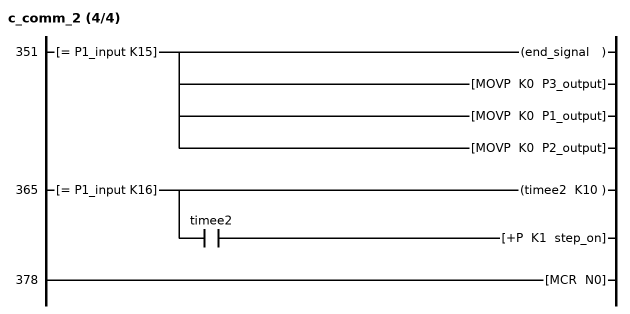
[picture p24: ladder of c_comm_2, rungs at steps 351 to 378]
351   LD=     P1_input K15
      OUT     end_signal
      MOVP    K0 P3_output
      MOVP    K0 P1_output
      MOVP    K0 P2_output
365   LD=     P1_input K16
      OUT     timee2 K10
      AND     timee2
      +P      K1 step_on
378   MCR     N0
END_FUNCTION_BLOCK

FUNCTION_BLOCK c_comm_3
VAR_INPUT
  P1_input : INT;
  P2_input : INT;
  P3_input : INT;
END_VAR
VAR_IN_OUT
  step_on : INT;
END_VAR
VAR_INPUT
  position : INT;
END_VAR
VAR
  p2_buff : INT;
END_VAR
VAR_OUTPUT
  P1_output : INT;
  P2_output : INT;
  P3_output : INT;
END_VAR
VAR_IN_OUT
  end_step_01 : INT;
END_VAR
VAR_OUTPUT
  end_signal : BOOL;
END_VAR
VAR
  mc_1234 : BOOL;
  line1_10_buff : INT;
  line2_10_buff : INT;
END_VAR
VAR_OUTPUT
  next_signal : BOOL;
END_VAR
VAR
  next_signal_01 : BOOL;
  next_signal_03 : BOOL;
  next_signal_04 : BOOL;
  next_signal_05 : BOOL;
  next_signal_06 : BOOL;
  next_signal_07 : BOOL;
  next_signal_08 : BOOL;
  punch1 : BOOL;
  punch3 : BOOL;
  punch4 : BOOL;
  punch5 : BOOL;
  punch6 : BOOL;
  punch7 : BOOL;
END_VAR
VAR_OUTPUT
  punch : BOOL;
END_VAR
VAR
  punch2 : BOOL;
  timee : TIMER;
  timee2 : TIMER;
END_VAR
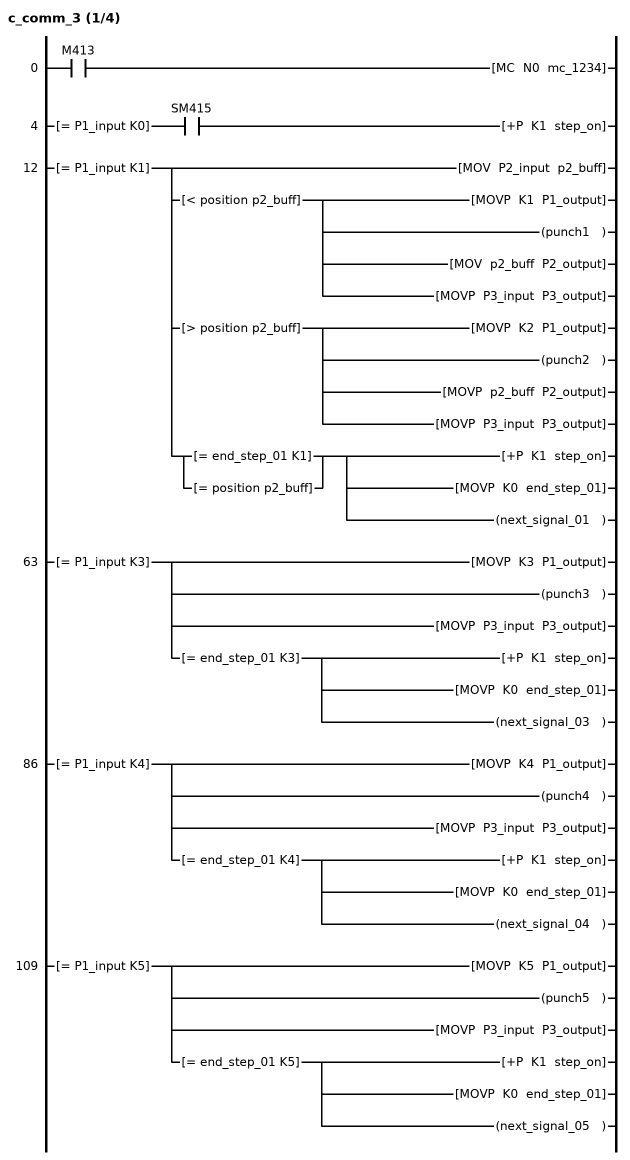
0     LD      M413
      MC      N0 mc_1234
4     LD=     P1_input K0
      AND     SM415
      +P      K1 step_on
12    LD=     P1_input K1
      MOV     P2_input p2_buff
      MPS
      AND<    position p2_buff
      MOVP    K1 P1_output
      OUT     punch1
      MOV     p2_buff P2_output
      MOVP    P3_input P3_output
      MRD
      AND>    position p2_buff
      MOVP    K2 P1_output
      OUT     punch2
      MOVP    p2_buff P2_output
      MOVP    P3_input P3_output
      MPP
      LD=     end_step_01 K1
      OR=     position p2_buff
      ANB
      +P      K1 step_on
      MOVP    K0 end_step_01
      OUT     next_signal_01
63    LD=     P1_input K3
      MOVP    K3 P1_output
      OUT     punch3
      MOVP    P3_input P3_output
      AND=    end_step_01 K3
      +P      K1 step_on
      MOVP    K0 end_step_01
      OUT     next_signal_03
86    LD=     P1_input K4
      MOVP    K4 P1_output
      OUT     punch4
      MOVP    P3_input P3_output
      AND=    end_step_01 K4
      +P      K1 step_on
      MOVP    K0 end_step_01
      OUT     next_signal_04
109   LD=     P1_input K5
      MOVP    K5 P1_output
      OUT     punch5
      MOVP    P3_input P3_output
      AND=    end_step_01 K5
      +P      K1 step_on
      MOVP    K0 end_step_01
      OUT     next_signal_05
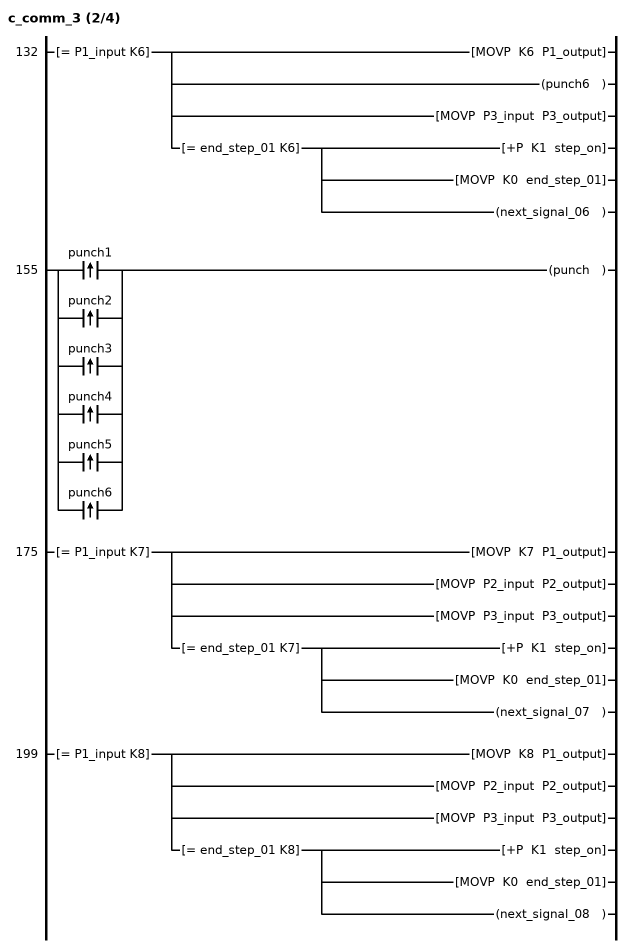
132   LD=     P1_input K6
      MOVP    K6 P1_output
      OUT     punch6
      MOVP    P3_input P3_output
      AND=    end_step_01 K6
      +P      K1 step_on
      MOVP    K0 end_step_01
      OUT     next_signal_06
155   LDP     punch1
      ORP     punch2
      ORP     punch3
      ORP     punch4
      ORP     punch5
      ORP     punch6
      OUT     punch
175   LD=     P1_input K7
      MOVP    K7 P1_output
      MOVP    P2_input P2_output
      MOVP    P3_input P3_output
      AND=    end_step_01 K7
      +P      K1 step_on
      MOVP    K0 end_step_01
      OUT     next_signal_07
199   LD=     P1_input K8
      MOVP    K8 P1_output
      MOVP    P2_input P2_output
      MOVP    P3_input P3_output
      AND=    end_step_01 K8
      +P      K1 step_on
      MOVP    K0 end_step_01
      OUT     next_signal_08
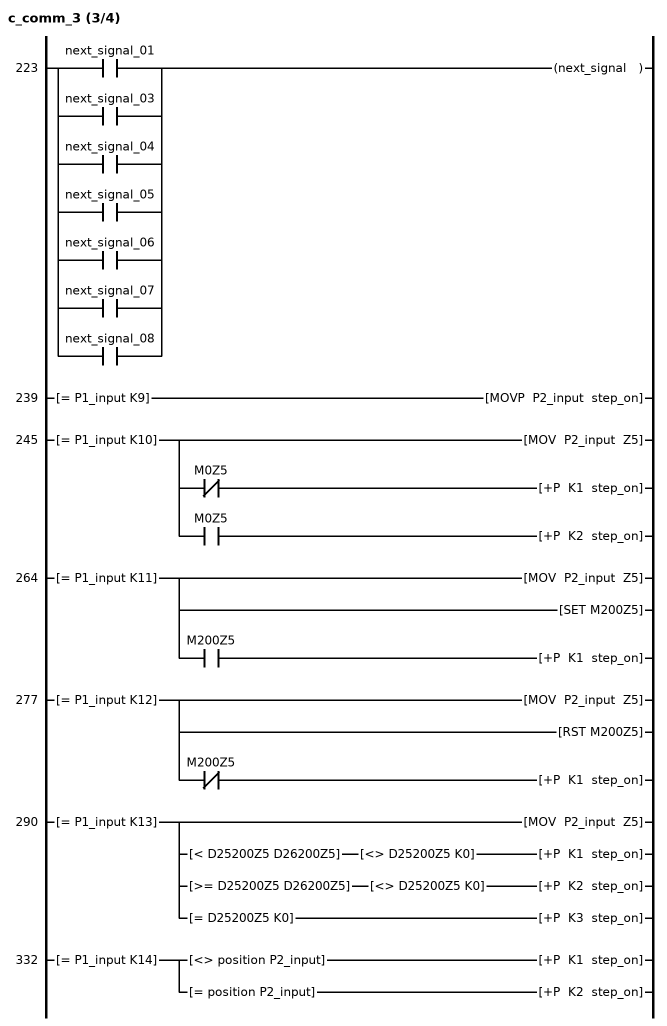
223   LD      next_signal_01
      OR      next_signal_03
      OR      next_signal_04
      OR      next_signal_05
      OR      next_signal_06
      OR      next_signal_07
      OR      next_signal_08
      OUT     next_signal
239   LD=     P1_input K9
      MOVP    P2_input step_on
245   LD=     P1_input K10
      MOV     P2_input Z5
      MPS
      ANI     M0Z5
      +P      K1 step_on
      MPP
      AND     M0Z5
      +P      K2 step_on
264   LD=     P1_input K11
      MOV     P2_input Z5
      SET     M200Z5
      AND     M200Z5
      +P      K1 step_on
277   LD=     P1_input K12
      MOV     P2_input Z5
      RST     M200Z5
      ANI     M200Z5
      +P      K1 step_on
290   LD=     P1_input K13
      MOV     P2_input Z5
      MPS
      AND<    D25200Z5 D26200Z5
      AND<>   D25200Z5 K0
      +P      K1 step_on
      MRD
      AND>=   D25200Z5 D26200Z5
      AND<>   D25200Z5 K0
      +P      K2 step_on
      MPP
      AND=    D25200Z5 K0
      +P      K3 step_on
332   LD=     P1_input K14
      MPS
      AND<>   position P2_input
      +P      K1 step_on
      MPP
      AND=    position P2_input
      +P      K2 step_on
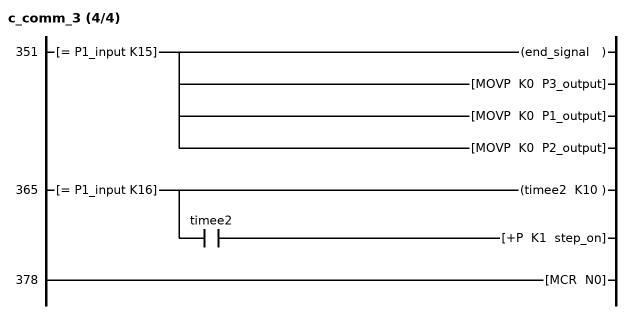
351   LD=     P1_input K15
      OUT     end_signal
      MOVP    K0 P3_output
      MOVP    K0 P1_output
      MOVP    K0 P2_output
365   LD=     P1_input K16
      OUT     timee2 K10
      AND     timee2
      +P      K1 step_on
378   MCR     N0
END_FUNCTION_BLOCK

PROGRAM carrier_01
VAR
  c_comm_1 : c_comm_1;
END_VAR
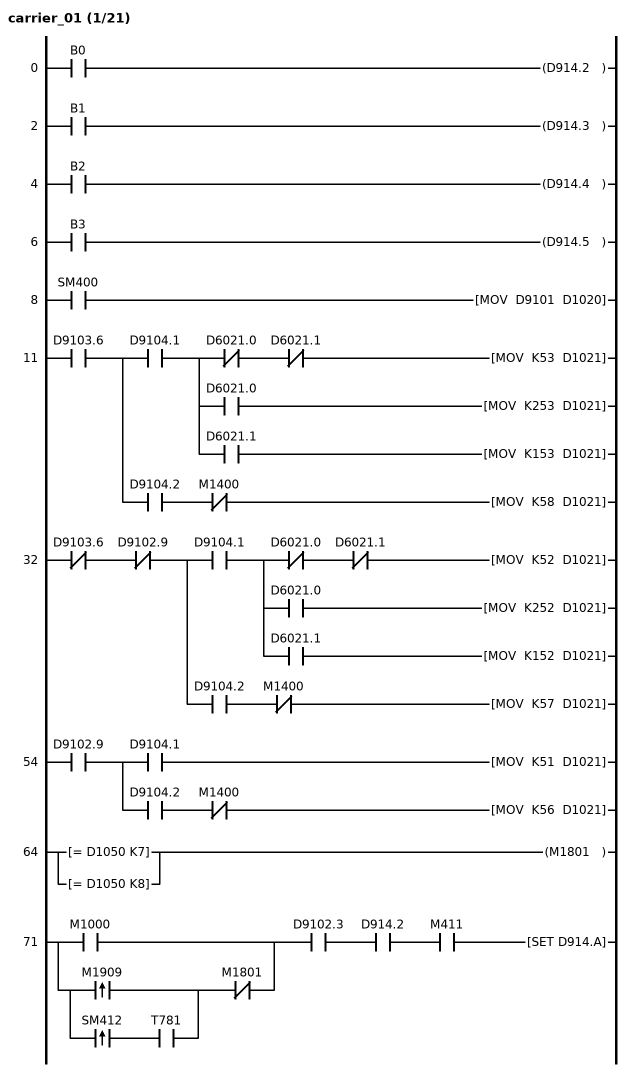
0     LD      B0
      OUT     D914.2
2     LD      B1
      OUT     D914.3
4     LD      B2
      OUT     D914.4
6     LD      B3
      OUT     D914.5
8     LD      SM400
      MOV     D9101 D1020
11    LD      D9103.6
      MPS
      AND     D9104.1
      MPS
      ANI     D6021.0
      ANI     D6021.1
      MOV     K53 D1021
      MRD
      AND     D6021.0
      MOV     K253 D1021
      MPP
      AND     D6021.1
      MOV     K153 D1021
      MPP
      AND     D9104.2
      ANI     M1400
      MOV     K58 D1021
32    LDI     D9103.6
      ANI     D9102.9
      MPS
      AND     D9104.1
      MPS
      ANI     D6021.0
      ANI     D6021.1
      MOV     K52 D1021
      MRD
      AND     D6021.0
      MOV     K252 D1021
      MPP
      AND     D6021.1
      MOV     K152 D1021
      MPP
      AND     D9104.2
      ANI     M1400
      MOV     K57 D1021
54    LD      D9102.9
      MPS
      AND     D9104.1
      MOV     K51 D1021
      MPP
      AND     D9104.2
      ANI     M1400
      MOV     K56 D1021
64    LD=     D1050 K7
      OR=     D1050 K8
      OUT     M1801
71    LD      M1000
      LDP     M1909
      LDP     SM412
      AND     T781
      ORB
      ANI     M1801
      ORB
      AND     D9102.3
      AND     D914.2
      AND     M411
      SET     D914.A
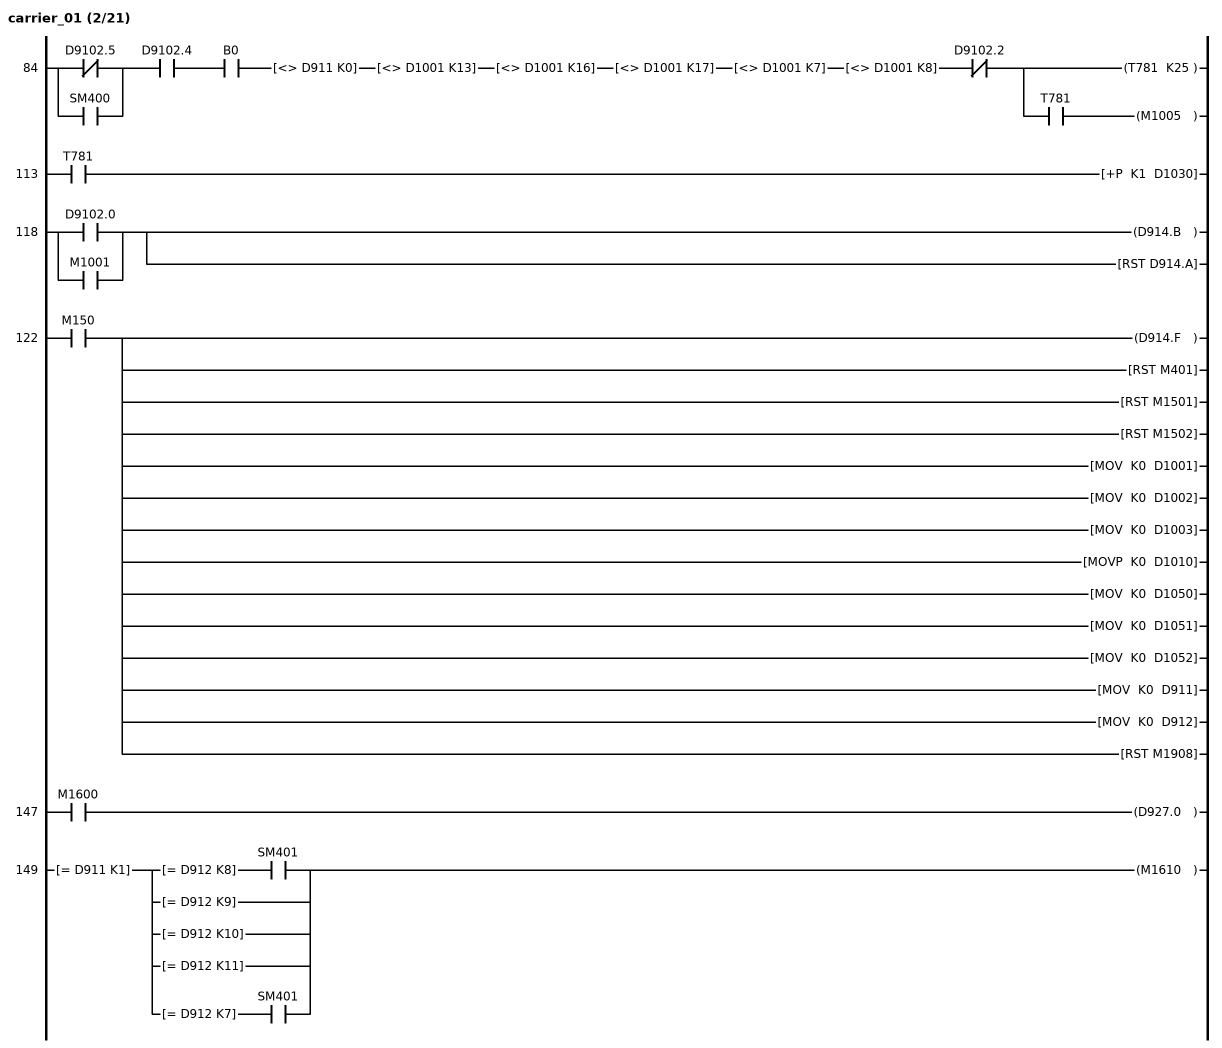
84    LDI     D9102.5
      OR      SM400
      AND     D9102.4
      AND     B0
      AND<>   D911 K0
      AND<>   D1001 K13
      AND<>   D1001 K16
      AND<>   D1001 K17
      AND<>   D1001 K7
      AND<>   D1001 K8
      ANI     D9102.2
      OUT     T781 K25
      AND     T781
      OUT     M1005
113   LD      T781
      +P      K1 D1030
118   LD      D9102.0
      OR      M1001
      OUT     D914.B
      RST     D914.A
122   LD      M150
      OUT     D914.F
      RST     M401
      RST     M1501
      RST     M1502
      MOV     K0 D1001
      MOV     K0 D1002
      MOV     K0 D1003
      MOVP    K0 D1010
      MOV     K0 D1050
      MOV     K0 D1051
      MOV     K0 D1052
      MOV     K0 D911
      MOV     K0 D912
      RST     M1908
147   LD      M1600
      OUT     D927.0
149   LD=     D911 K1
      LD=     D912 K8
      AND     SM401
      OR=     D912 K9
      OR=     D912 K10
      OR=     D912 K11
      LD=     D912 K7
      AND     SM401
      ORB
      ANB
      OUT     M1610
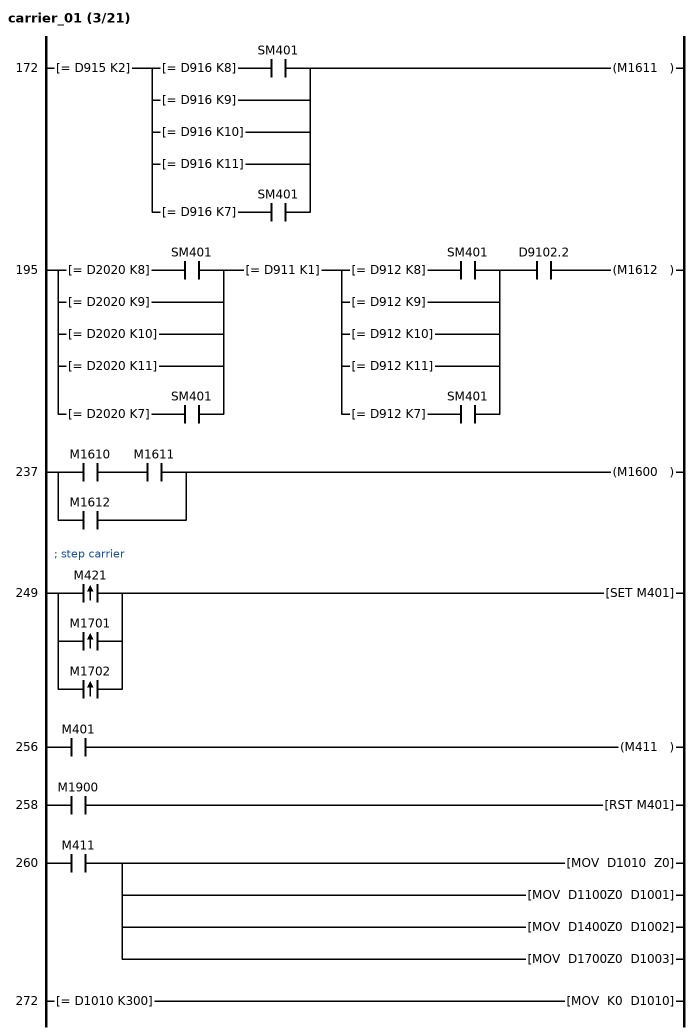
172   LD=     D915 K2
      LD=     D916 K8
      AND     SM401
      OR=     D916 K9
      OR=     D916 K10
      OR=     D916 K11
      LD=     D916 K7
      AND     SM401
      ORB
      ANB
      OUT     M1611
195   LD=     D2020 K8
      AND     SM401
      OR=     D2020 K9
      OR=     D2020 K10
      OR=     D2020 K11
      LD=     D2020 K7
      AND     SM401
      ORB
      AND=    D911 K1
      LD=     D912 K8
      AND     SM401
      OR=     D912 K9
      OR=     D912 K10
      OR=     D912 K11
      LD=     D912 K7
      AND     SM401
      ORB
      ANB
      AND     D9102.2
      OUT     M1612
237   LD      M1610
      AND     M1611
      OR      M1612
      OUT     M1600
; step carrier
249   LDP     M421
      ORP     M1701
      ORP     M1702
      SET     M401
256   LD      M401
      OUT     M411
258   LD      M1900
      RST     M401
260   LD      M411
      MOV     D1010 Z0
      MOV     D1100Z0 D1001
      MOV     D1400Z0 D1002
      MOV     D1700Z0 D1003
272   LD=     D1010 K300
      MOV     K0 D1010
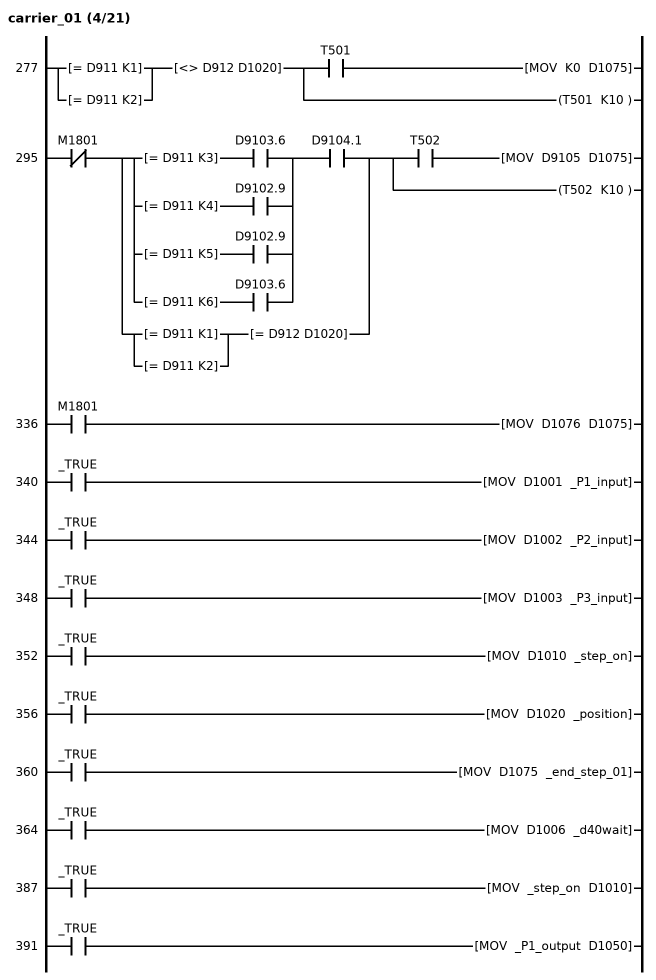
277   LD=     D911 K1
      OR=     D911 K2
      AND<>   D912 D1020
      MPS
      AND     T501
      MOV     K0 D1075
      MPP
      OUT     T501 K10
295   LDI     M1801
      LD=     D911 K3
      AND     D9103.6
      LD=     D911 K4
      AND     D9102.9
      ORB
      LD=     D911 K5
      AND     D9102.9
      ORB
      LD=     D911 K6
      AND     D9103.6
      ORB
      AND     D9104.1
      LD=     D911 K1
      OR=     D911 K2
      AND=    D912 D1020
      ORB
      ANB
      MPS
      AND     T502
      MOV     D9105 D1075
      MPP
      OUT     T502 K10
336   LD      M1801
      MOV     D1076 D1075
; FB BLK START c_comm_1(c_comm_1)
340   LD      _TRUE
      MOV     D1001 _P1_input
344   LD      _TRUE
      MOV     D1002 _P2_input
348   LD      _TRUE
      MOV     D1003 _P3_input
352   LD      _TRUE
      MOV     D1010 _step_on
356   LD      _TRUE
      MOV     D1020 _position
360   LD      _TRUE
      MOV     D1075 _end_step_01
364   LD      _TRUE
      MOV     D1006 _d40wait
; FB START
; FB_NAME c_comm_1
; INSTANCE_NAME c_comm_1
; FB IN_W:P1_input
; FB OUT_step_on:W
; FB IN_W:P2_input
; FB OUT_P1_output:W
; FB IN_W:P3_input
; FB OUT_P2_output:W
; FB IN_W:step_on
; FB OUT_P3_output:W
; FB IN_W:position
; FB OUT_end_step_01:W
; FB IN_W:end_step_01
; FB OUT_end_signal:B
; FB IN_W:d40wait
; FB OUT_next_signal:B
; FB OUT_punch:B
; FB END
387   LD      _TRUE
      MOV     _step_on D1010
391   LD      _TRUE
      MOV     _P1_output D1050
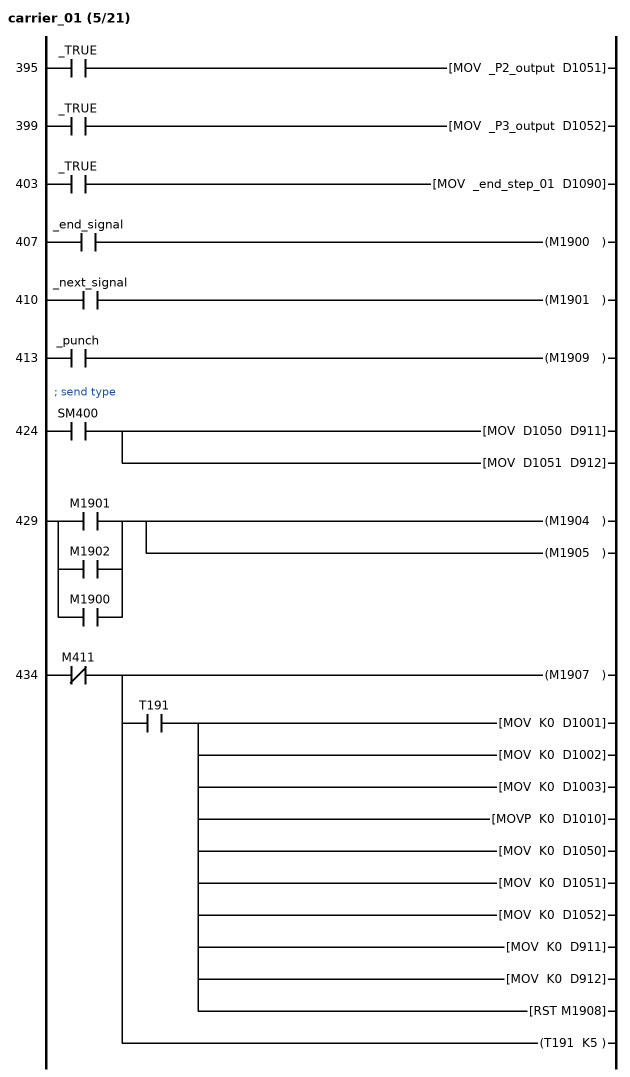
395   LD      _TRUE
      MOV     _P2_output D1051
399   LD      _TRUE
      MOV     _P3_output D1052
403   LD      _TRUE
      MOV     _end_step_01 D1090
407   LD      _end_signal
      OUT     M1900
410   LD      _next_signal
      OUT     M1901
413   LD      _punch
      OUT     M1909
; FB BLK END
; send type
424   LD      SM400
      MOV     D1050 D911
      MOV     D1051 D912
429   LD      M1901
      OR      M1902
      OR      M1900
      OUT     M1904
      OUT     M1905
434   LDI     M411
      OUT     M1907
      MPS
      AND     T191
      MOV     K0 D1001
      MOV     K0 D1002
      MOV     K0 D1003
      MOVP    K0 D1010
      MOV     K0 D1050
      MOV     K0 D1051
      MOV     K0 D1052
      MOV     K0 D911
      MOV     K0 D912
      RST     M1908
      MPP
      OUT     T191 K5
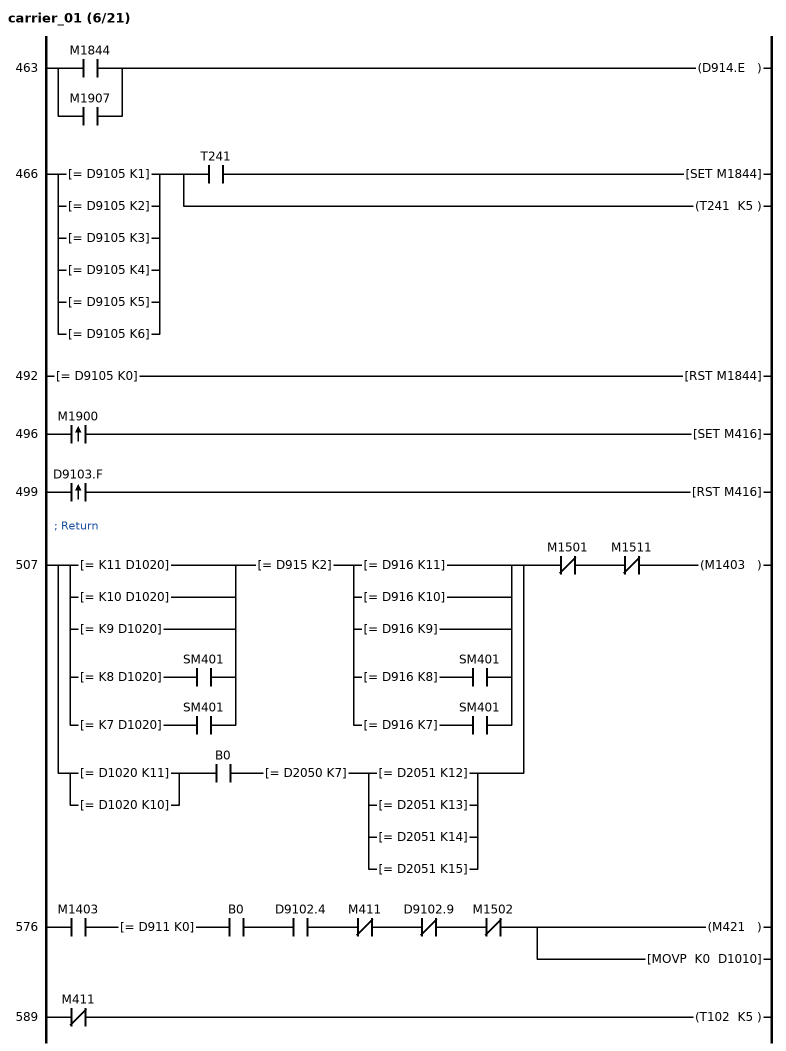
463   LD      M1844
      OR      M1907
      OUT     D914.E
466   LD=     D9105 K1
      OR=     D9105 K2
      OR=     D9105 K3
      OR=     D9105 K4
      OR=     D9105 K5
      OR=     D9105 K6
      MPS
      AND     T241
      SET     M1844
      MPP
      OUT     T241 K5
492   LD=     D9105 K0
      RST     M1844
496   LDP     M1900
      SET     M416
499   LDP     D9103.F
      RST     M416
; Return
507   LD=     K11 D1020
      OR=     K10 D1020
      OR=     K9 D1020
      LD=     K8 D1020
      AND     SM401
      ORB
      LD=     K7 D1020
      AND     SM401
      ORB
      AND=    D915 K2
      LD=     D916 K11
      OR=     D916 K10
      OR=     D916 K9
      LD=     D916 K8
      AND     SM401
      ORB
      LD=     D916 K7
      AND     SM401
      ORB
      ANB
      LD=     D1020 K11
      OR=     D1020 K10
      AND     B0
      AND=    D2050 K7
      LD=     D2051 K12
      OR=     D2051 K13
      OR=     D2051 K14
      OR=     D2051 K15
      ANB
      ORB
      ANI     M1501
      ANI     M1511
      OUT     M1403
576   LD      M1403
      AND=    D911 K0
      AND     B0
      AND     D9102.4
      ANI     M411
      ANI     D9102.9
      ANI     M1502
      OUT     M421
      MOVP    K0 D1010
589   LDI     M411
      OUT     T102 K5
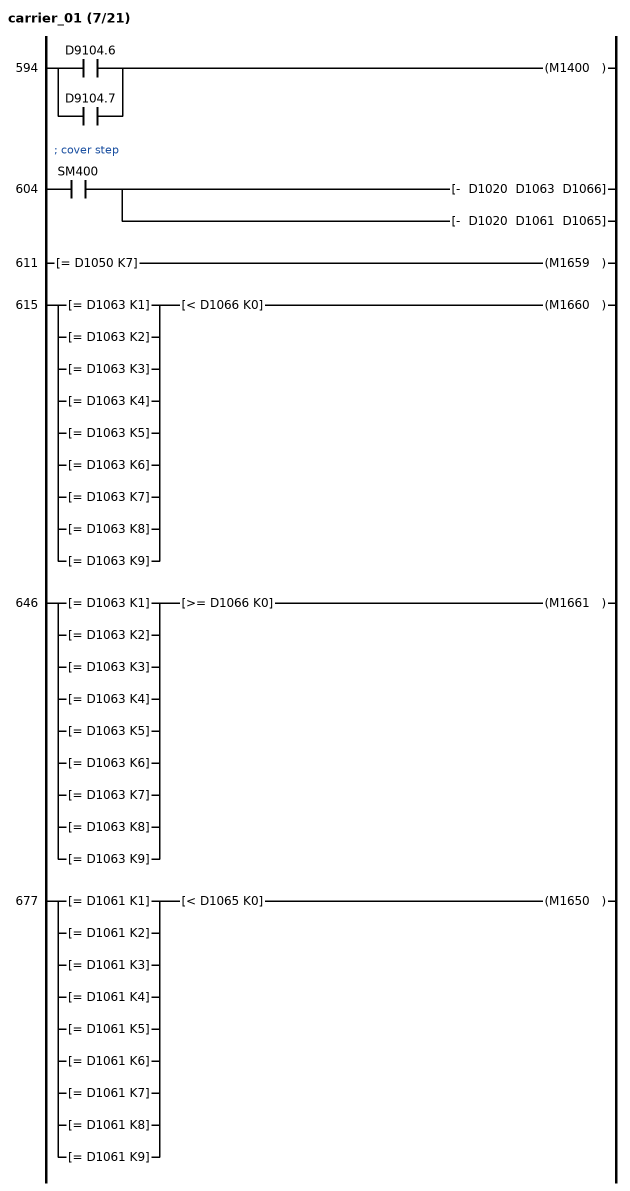
594   LD      D9104.6
      OR      D9104.7
      OUT     M1400
; cover step
604   LD      SM400
      -       D1020 D1063 D1066
      -       D1020 D1061 D1065
611   LD=     D1050 K7
      OUT     M1659
615   LD=     D1063 K1
      OR=     D1063 K2
      OR=     D1063 K3
      OR=     D1063 K4
      OR=     D1063 K5
      OR=     D1063 K6
      OR=     D1063 K7
      OR=     D1063 K8
      OR=     D1063 K9
      AND<    D1066 K0
      OUT     M1660
646   LD=     D1063 K1
      OR=     D1063 K2
      OR=     D1063 K3
      OR=     D1063 K4
      OR=     D1063 K5
      OR=     D1063 K6
      OR=     D1063 K7
      OR=     D1063 K8
      OR=     D1063 K9
      AND>=   D1066 K0
      OUT     M1661
677   LD=     D1061 K1
      OR=     D1061 K2
      OR=     D1061 K3
      OR=     D1061 K4
      OR=     D1061 K5
      OR=     D1061 K6
      OR=     D1061 K7
      OR=     D1061 K8
      OR=     D1061 K9
      AND<    D1065 K0
      OUT     M1650
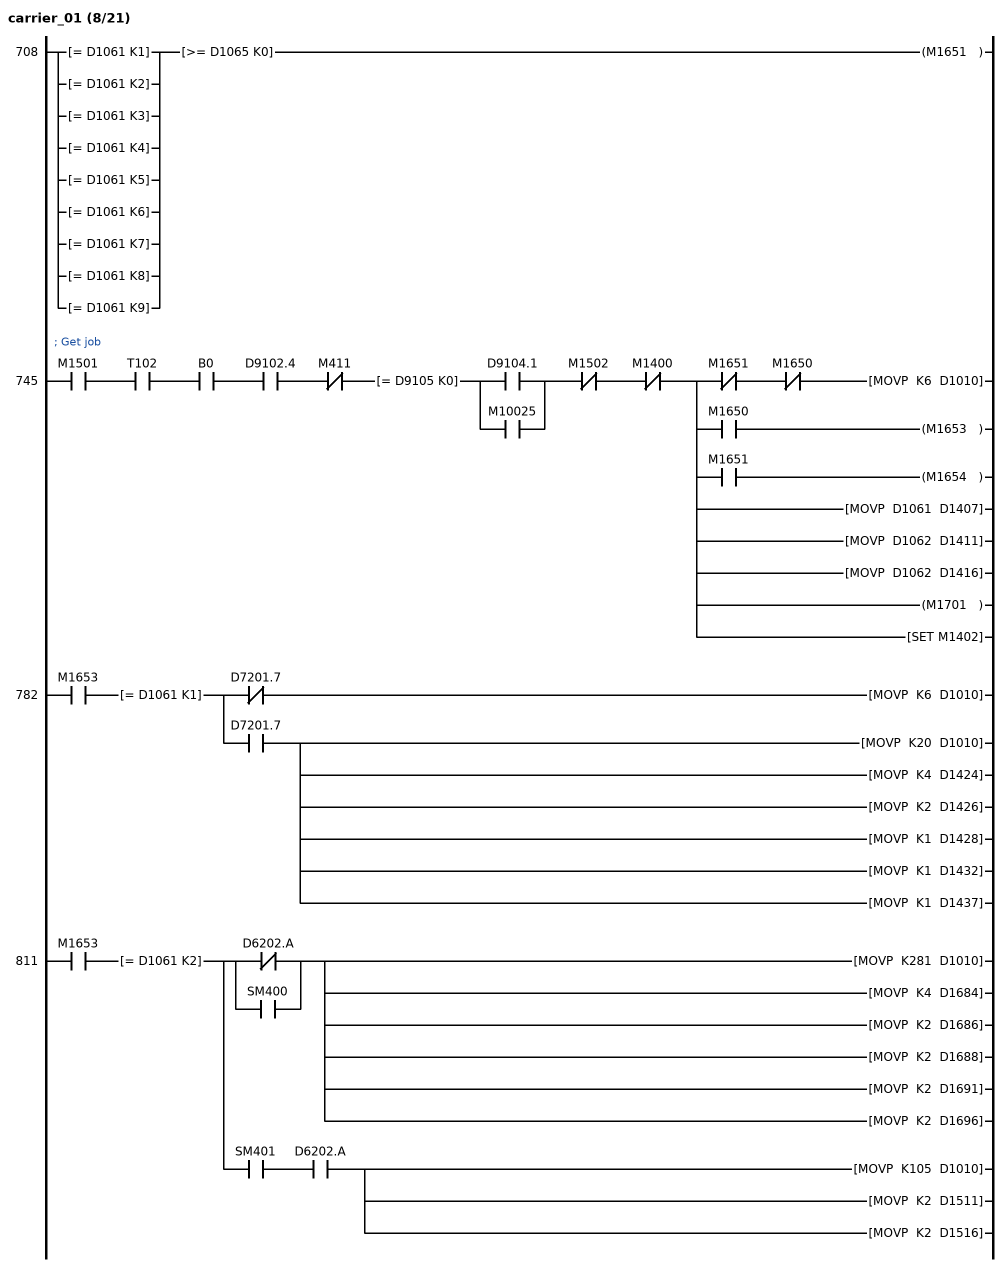
708   LD=     D1061 K1
      OR=     D1061 K2
      OR=     D1061 K3
      OR=     D1061 K4
      OR=     D1061 K5
      OR=     D1061 K6
      OR=     D1061 K7
      OR=     D1061 K8
      OR=     D1061 K9
      AND>=   D1065 K0
      OUT     M1651
; Get job
745   LD      M1501
      AND     T102
      AND     B0
      AND     D9102.4
      ANI     M411
      AND=    D9105 K0
      LD      D9104.1
      OR      M10025
      ANB
      ANI     M1502
      ANI     M1400
      MPS
      ANI     M1651
      ANI     M1650
      MOVP    K6 D1010
      MRD
      AND     M1650
      OUT     M1653
      MRD
      AND     M1651
      OUT     M1654
      MPP
      MOVP    D1061 D1407
      MOVP    D1062 D1411
      MOVP    D1062 D1416
      OUT     M1701
      SET     M1402
782   LD      M1653
      AND=    D1061 K1
      MPS
      ANI     D7201.7
      MOVP    K6 D1010
      MPP
      AND     D7201.7
      MOVP    K20 D1010
      MOVP    K4 D1424
      MOVP    K2 D1426
      MOVP    K1 D1428
      MOVP    K1 D1432
      MOVP    K1 D1437
811   LD      M1653
      AND=    D1061 K2
      MPS
      LDI     D6202.A
      OR      SM400
      ANB
      MOVP    K281 D1010
      MOVP    K4 D1684
      MOVP    K2 D1686
      MOVP    K2 D1688
      MOVP    K2 D1691
      MOVP    K2 D1696
      MPP
      AND     SM401
      AND     D6202.A
      MOVP    K105 D1010
      MOVP    K2 D1511
      MOVP    K2 D1516
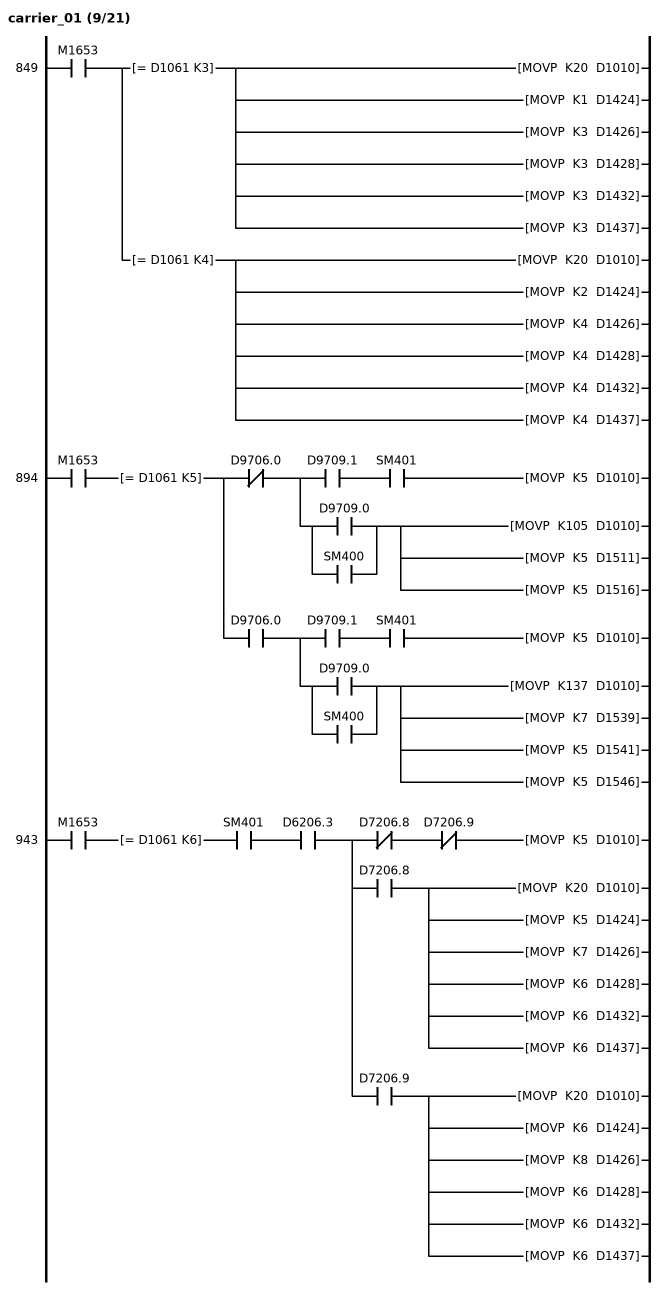
849   LD      M1653
      MPS
      AND=    D1061 K3
      MOVP    K20 D1010
      MOVP    K1 D1424
      MOVP    K3 D1426
      MOVP    K3 D1428
      MOVP    K3 D1432
      MOVP    K3 D1437
      MPP
      AND=    D1061 K4
      MOVP    K20 D1010
      MOVP    K2 D1424
      MOVP    K4 D1426
      MOVP    K4 D1428
      MOVP    K4 D1432
      MOVP    K4 D1437
894   LD      M1653
      AND=    D1061 K5
      MPS
      ANI     D9706.0
      MPS
      AND     D9709.1
      AND     SM401
      MOVP    K5 D1010
      MPP
      LD      D9709.0
      OR      SM400
      ANB
      MOVP    K105 D1010
      MOVP    K5 D1511
      MOVP    K5 D1516
      MPP
      AND     D9706.0
      MPS
      AND     D9709.1
      AND     SM401
      MOVP    K5 D1010
      MPP
      LD      D9709.0
      OR      SM400
      ANB
      MOVP    K137 D1010
      MOVP    K7 D1539
      MOVP    K5 D1541
      MOVP    K5 D1546
943   LD      M1653
      AND=    D1061 K6
      AND     SM401
      AND     D6206.3
      MPS
      ANI     D7206.8
      ANI     D7206.9
      MOVP    K5 D1010
      MRD
      AND     D7206.8
      MOVP    K20 D1010
      MOVP    K5 D1424
      MOVP    K7 D1426
      MOVP    K6 D1428
      MOVP    K6 D1432
      MOVP    K6 D1437
      MPP
      AND     D7206.9
      MOVP    K20 D1010
      MOVP    K6 D1424
      MOVP    K8 D1426
      MOVP    K6 D1428
      MOVP    K6 D1432
      MOVP    K6 D1437
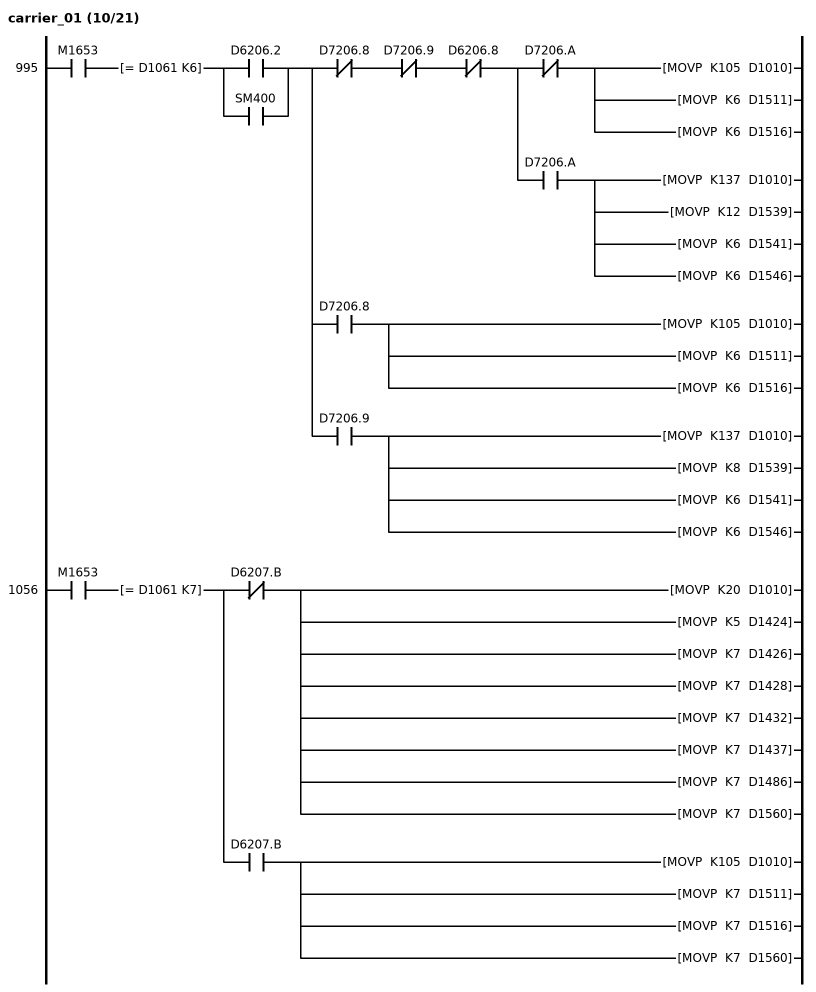
995   LD      M1653
      AND=    D1061 K6
      LD      D6206.2
      OR      SM400
      ANB
      MPS
      ANI     D7206.8
      ANI     D7206.9
      ANI     D6206.8
      MPS
      ANI     D7206.A
      MOVP    K105 D1010
      MOVP    K6 D1511
      MOVP    K6 D1516
      MPP
      AND     D7206.A
      MOVP    K137 D1010
      MOVP    K12 D1539
      MOVP    K6 D1541
      MOVP    K6 D1546
      MRD
      AND     D7206.8
      MOVP    K105 D1010
      MOVP    K6 D1511
      MOVP    K6 D1516
      MPP
      AND     D7206.9
      MOVP    K137 D1010
      MOVP    K8 D1539
      MOVP    K6 D1541
      MOVP    K6 D1546
1056  LD      M1653
      AND=    D1061 K7
      MPS
      ANI     D6207.B
      MOVP    K20 D1010
      MOVP    K5 D1424
      MOVP    K7 D1426
      MOVP    K7 D1428
      MOVP    K7 D1432
      MOVP    K7 D1437
      MOVP    K7 D1486
      MOVP    K7 D1560
      MPP
      AND     D6207.B
      MOVP    K105 D1010
      MOVP    K7 D1511
      MOVP    K7 D1516
      MOVP    K7 D1560
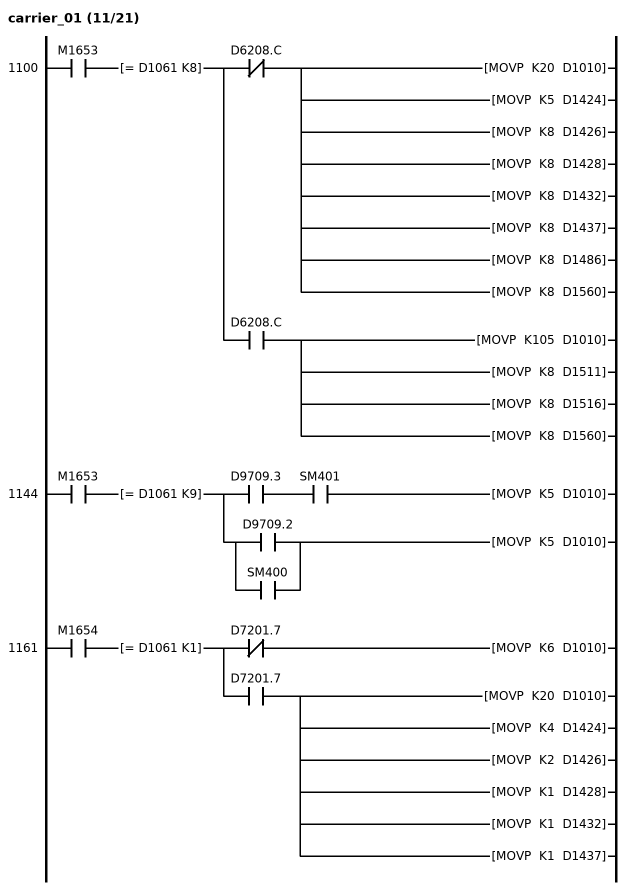
1100  LD      M1653
      AND=    D1061 K8
      MPS
      ANI     D6208.C
      MOVP    K20 D1010
      MOVP    K5 D1424
      MOVP    K8 D1426
      MOVP    K8 D1428
      MOVP    K8 D1432
      MOVP    K8 D1437
      MOVP    K8 D1486
      MOVP    K8 D1560
      MPP
      AND     D6208.C
      MOVP    K105 D1010
      MOVP    K8 D1511
      MOVP    K8 D1516
      MOVP    K8 D1560
1144  LD      M1653
      AND=    D1061 K9
      MPS
      AND     D9709.3
      AND     SM401
      MOVP    K5 D1010
      MPP
      LD      D9709.2
      OR      SM400
      ANB
      MOVP    K5 D1010
1161  LD      M1654
      AND=    D1061 K1
      MPS
      ANI     D7201.7
      MOVP    K6 D1010
      MPP
      AND     D7201.7
      MOVP    K20 D1010
      MOVP    K4 D1424
      MOVP    K2 D1426
      MOVP    K1 D1428
      MOVP    K1 D1432
      MOVP    K1 D1437
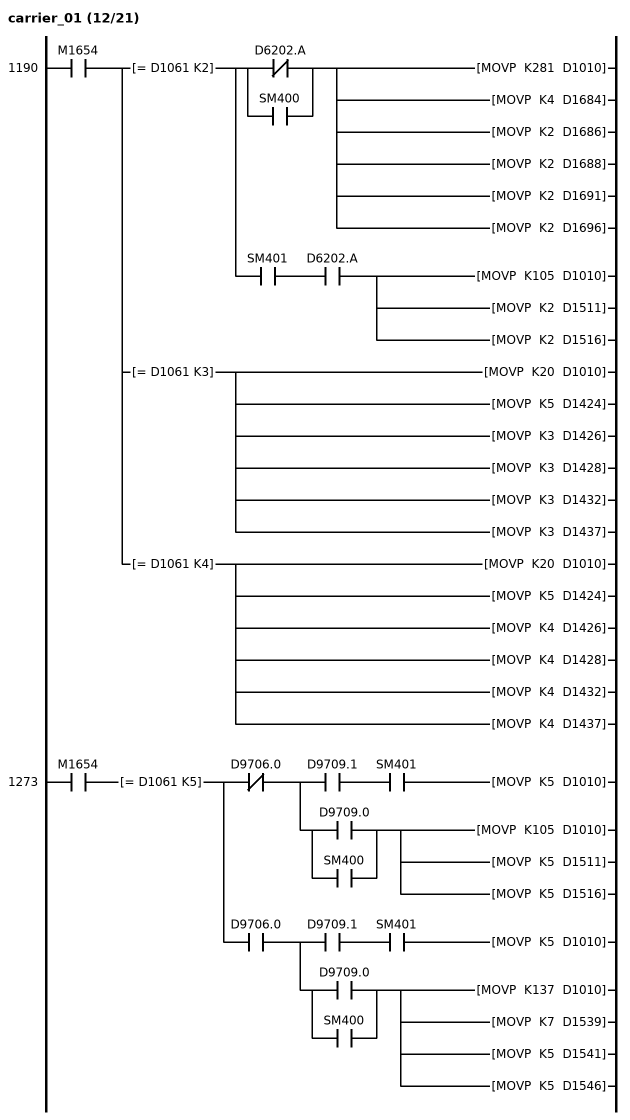
1190  LD      M1654
      MPS
      AND=    D1061 K2
      MPS
      LDI     D6202.A
      OR      SM400
      ANB
      MOVP    K281 D1010
      MOVP    K4 D1684
      MOVP    K2 D1686
      MOVP    K2 D1688
      MOVP    K2 D1691
      MOVP    K2 D1696
      MPP
      AND     SM401
      AND     D6202.A
      MOVP    K105 D1010
      MOVP    K2 D1511
      MOVP    K2 D1516
      MRD
      AND=    D1061 K3
      MOVP    K20 D1010
      MOVP    K5 D1424
      MOVP    K3 D1426
      MOVP    K3 D1428
      MOVP    K3 D1432
      MOVP    K3 D1437
      MPP
      AND=    D1061 K4
      MOVP    K20 D1010
      MOVP    K5 D1424
      MOVP    K4 D1426
      MOVP    K4 D1428
      MOVP    K4 D1432
      MOVP    K4 D1437
1273  LD      M1654
      AND=    D1061 K5
      MPS
      ANI     D9706.0
      MPS
      AND     D9709.1
      AND     SM401
      MOVP    K5 D1010
      MPP
      LD      D9709.0
      OR      SM400
      ANB
      MOVP    K105 D1010
      MOVP    K5 D1511
      MOVP    K5 D1516
      MPP
      AND     D9706.0
      MPS
      AND     D9709.1
      AND     SM401
      MOVP    K5 D1010
      MPP
      LD      D9709.0
      OR      SM400
      ANB
      MOVP    K137 D1010
      MOVP    K7 D1539
      MOVP    K5 D1541
      MOVP    K5 D1546
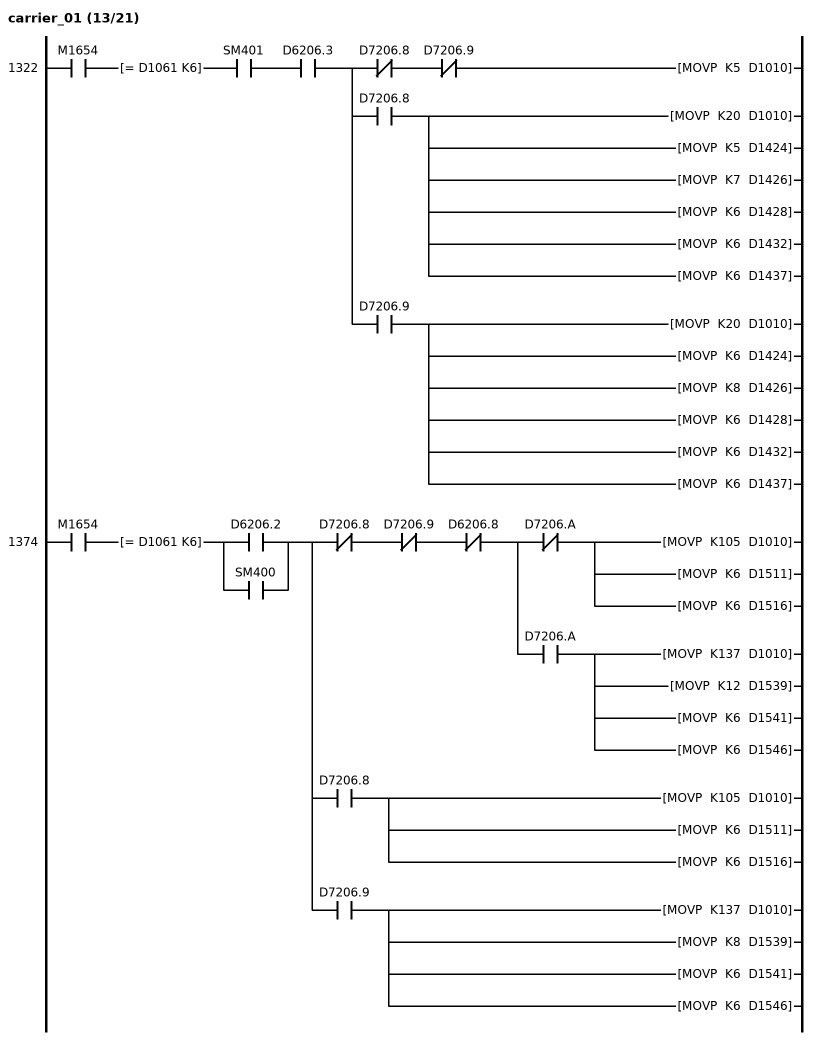
1322  LD      M1654
      AND=    D1061 K6
      AND     SM401
      AND     D6206.3
      MPS
      ANI     D7206.8
      ANI     D7206.9
      MOVP    K5 D1010
      MRD
      AND     D7206.8
      MOVP    K20 D1010
      MOVP    K5 D1424
      MOVP    K7 D1426
      MOVP    K6 D1428
      MOVP    K6 D1432
      MOVP    K6 D1437
      MPP
      AND     D7206.9
      MOVP    K20 D1010
      MOVP    K6 D1424
      MOVP    K8 D1426
      MOVP    K6 D1428
      MOVP    K6 D1432
      MOVP    K6 D1437
1374  LD      M1654
      AND=    D1061 K6
      LD      D6206.2
      OR      SM400
      ANB
      MPS
      ANI     D7206.8
      ANI     D7206.9
      ANI     D6206.8
      MPS
      ANI     D7206.A
      MOVP    K105 D1010
      MOVP    K6 D1511
      MOVP    K6 D1516
      MPP
      AND     D7206.A
      MOVP    K137 D1010
      MOVP    K12 D1539
      MOVP    K6 D1541
      MOVP    K6 D1546
      MRD
      AND     D7206.8
      MOVP    K105 D1010
      MOVP    K6 D1511
      MOVP    K6 D1516
      MPP
      AND     D7206.9
      MOVP    K137 D1010
      MOVP    K8 D1539
      MOVP    K6 D1541
      MOVP    K6 D1546
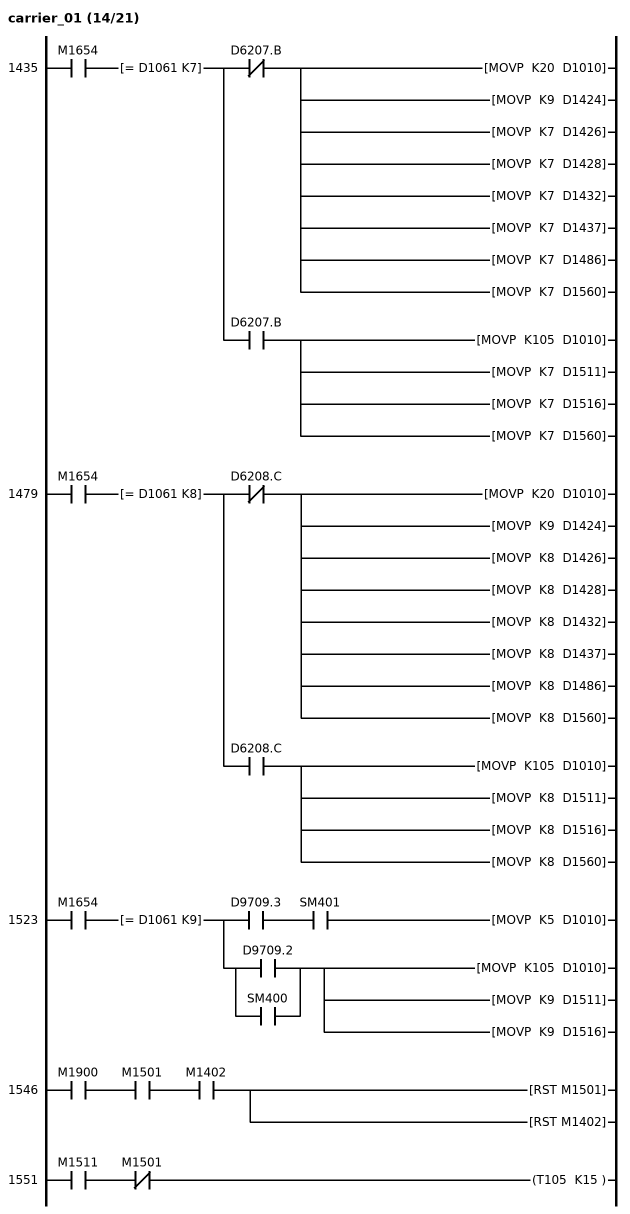
1435  LD      M1654
      AND=    D1061 K7
      MPS
      ANI     D6207.B
      MOVP    K20 D1010
      MOVP    K9 D1424
      MOVP    K7 D1426
      MOVP    K7 D1428
      MOVP    K7 D1432
      MOVP    K7 D1437
      MOVP    K7 D1486
      MOVP    K7 D1560
      MPP
      AND     D6207.B
      MOVP    K105 D1010
      MOVP    K7 D1511
      MOVP    K7 D1516
      MOVP    K7 D1560
1479  LD      M1654
      AND=    D1061 K8
      MPS
      ANI     D6208.C
      MOVP    K20 D1010
      MOVP    K9 D1424
      MOVP    K8 D1426
      MOVP    K8 D1428
      MOVP    K8 D1432
      MOVP    K8 D1437
      MOVP    K8 D1486
      MOVP    K8 D1560
      MPP
      AND     D6208.C
      MOVP    K105 D1010
      MOVP    K8 D1511
      MOVP    K8 D1516
      MOVP    K8 D1560
1523  LD      M1654
      AND=    D1061 K9
      MPS
      AND     D9709.3
      AND     SM401
      MOVP    K5 D1010
      MPP
      LD      D9709.2
      OR      SM400
      ANB
      MOVP    K105 D1010
      MOVP    K9 D1511
      MOVP    K9 D1516
1546  LD      M1900
      AND     M1501
      AND     M1402
      RST     M1501
      RST     M1402
1551  LD      M1511
      ANI     M1501
      OUT     T105 K15
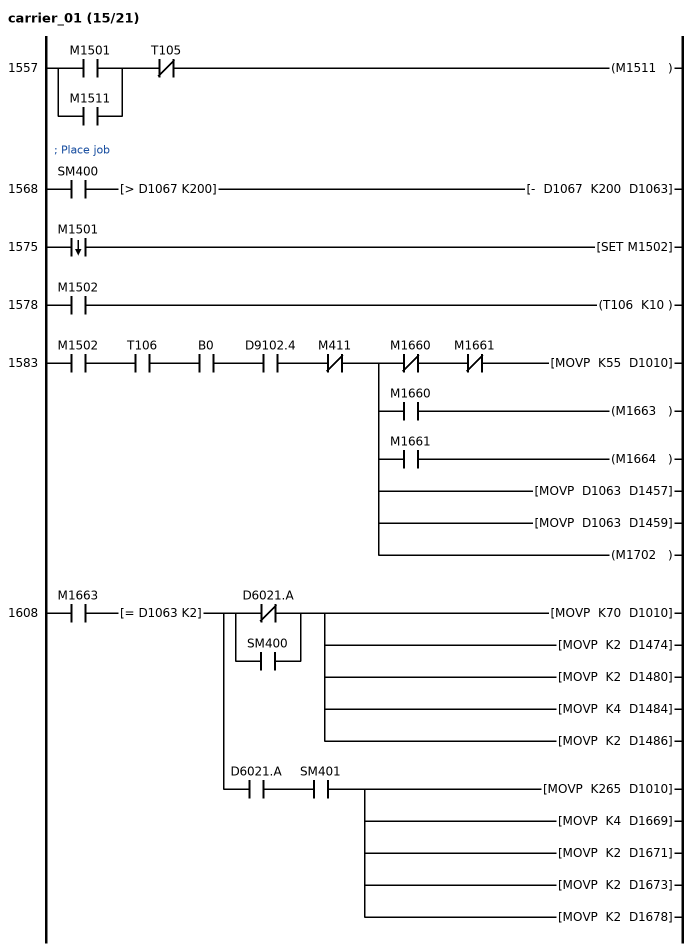
1557  LD      M1501
      OR      M1511
      ANI     T105
      OUT     M1511
; Place job
1568  LD      SM400
      AND>    D1067 K200
      -       D1067 K200 D1063
1575  LDF     M1501
      SET     M1502
1578  LD      M1502
      OUT     T106 K10
1583  LD      M1502
      AND     T106
      AND     B0
      AND     D9102.4
      ANI     M411
      MPS
      ANI     M1660
      ANI     M1661
      MOVP    K55 D1010
      MRD
      AND     M1660
      OUT     M1663
      MRD
      AND     M1661
      OUT     M1664
      MPP
      MOVP    D1063 D1457
      MOVP    D1063 D1459
      OUT     M1702
1608  LD      M1663
      AND=    D1063 K2
      MPS
      LDI     D6021.A
      OR      SM400
      ANB
      MOVP    K70 D1010
      MOVP    K2 D1474
      MOVP    K2 D1480
      MOVP    K4 D1484
      MOVP    K2 D1486
      MPP
      AND     D6021.A
      AND     SM401
      MOVP    K265 D1010
      MOVP    K4 D1669
      MOVP    K2 D1671
      MOVP    K2 D1673
      MOVP    K2 D1678
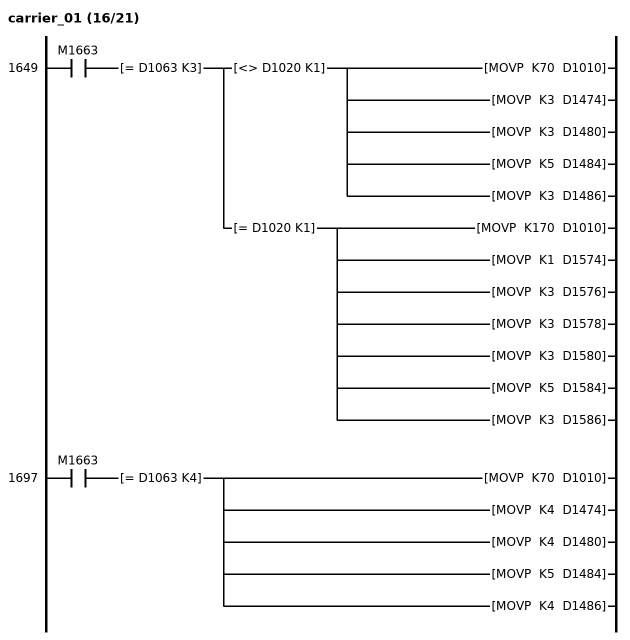
1649  LD      M1663
      AND=    D1063 K3
      MPS
      AND<>   D1020 K1
      MOVP    K70 D1010
      MOVP    K3 D1474
      MOVP    K3 D1480
      MOVP    K5 D1484
      MOVP    K3 D1486
      MPP
      AND=    D1020 K1
      MOVP    K170 D1010
      MOVP    K1 D1574
      MOVP    K3 D1576
      MOVP    K3 D1578
      MOVP    K3 D1580
      MOVP    K5 D1584
      MOVP    K3 D1586
1697  LD      M1663
      AND=    D1063 K4
      MOVP    K70 D1010
      MOVP    K4 D1474
      MOVP    K4 D1480
      MOVP    K5 D1484
      MOVP    K4 D1486
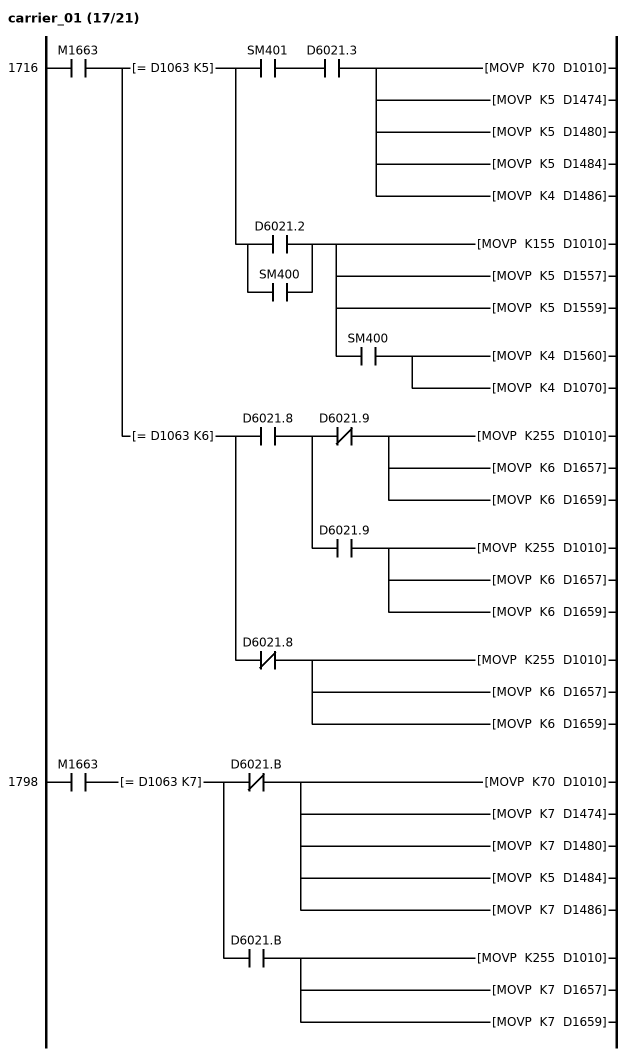
1716  LD      M1663
      MPS
      AND=    D1063 K5
      MPS
      AND     SM401
      AND     D6021.3
      MOVP    K70 D1010
      MOVP    K5 D1474
      MOVP    K5 D1480
      MOVP    K5 D1484
      MOVP    K4 D1486
      MPP
      LD      D6021.2
      OR      SM400
      ANB
      MOVP    K155 D1010
      MOVP    K5 D1557
      MOVP    K5 D1559
      AND     SM400
      MOVP    K4 D1560
      MOVP    K4 D1070
      MPP
      AND=    D1063 K6
      MPS
      AND     D6021.8
      MPS
      ANI     D6021.9
      MOVP    K255 D1010
      MOVP    K6 D1657
      MOVP    K6 D1659
      MPP
      AND     D6021.9
      MOVP    K255 D1010
      MOVP    K6 D1657
      MOVP    K6 D1659
      MPP
      ANI     D6021.8
      MOVP    K255 D1010
      MOVP    K6 D1657
      MOVP    K6 D1659
1798  LD      M1663
      AND=    D1063 K7
      MPS
      ANI     D6021.B
      MOVP    K70 D1010
      MOVP    K7 D1474
      MOVP    K7 D1480
      MOVP    K5 D1484
      MOVP    K7 D1486
      MPP
      AND     D6021.B
      MOVP    K255 D1010
      MOVP    K7 D1657
      MOVP    K7 D1659
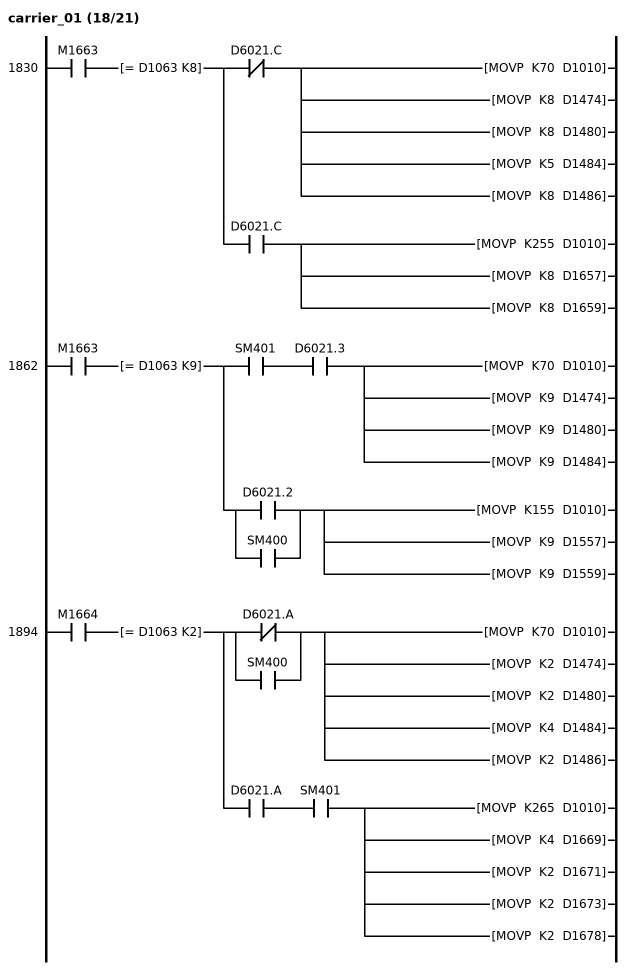
1830  LD      M1663
      AND=    D1063 K8
      MPS
      ANI     D6021.C
      MOVP    K70 D1010
      MOVP    K8 D1474
      MOVP    K8 D1480
      MOVP    K5 D1484
      MOVP    K8 D1486
      MPP
      AND     D6021.C
      MOVP    K255 D1010
      MOVP    K8 D1657
      MOVP    K8 D1659
1862  LD      M1663
      AND=    D1063 K9
      MPS
      AND     SM401
      AND     D6021.3
      MOVP    K70 D1010
      MOVP    K9 D1474
      MOVP    K9 D1480
      MOVP    K9 D1484
      MPP
      LD      D6021.2
      OR      SM400
      ANB
      MOVP    K155 D1010
      MOVP    K9 D1557
      MOVP    K9 D1559
1894  LD      M1664
      AND=    D1063 K2
      MPS
      LDI     D6021.A
      OR      SM400
      ANB
      MOVP    K70 D1010
      MOVP    K2 D1474
      MOVP    K2 D1480
      MOVP    K4 D1484
      MOVP    K2 D1486
      MPP
      AND     D6021.A
      AND     SM401
      MOVP    K265 D1010
      MOVP    K4 D1669
      MOVP    K2 D1671
      MOVP    K2 D1673
      MOVP    K2 D1678
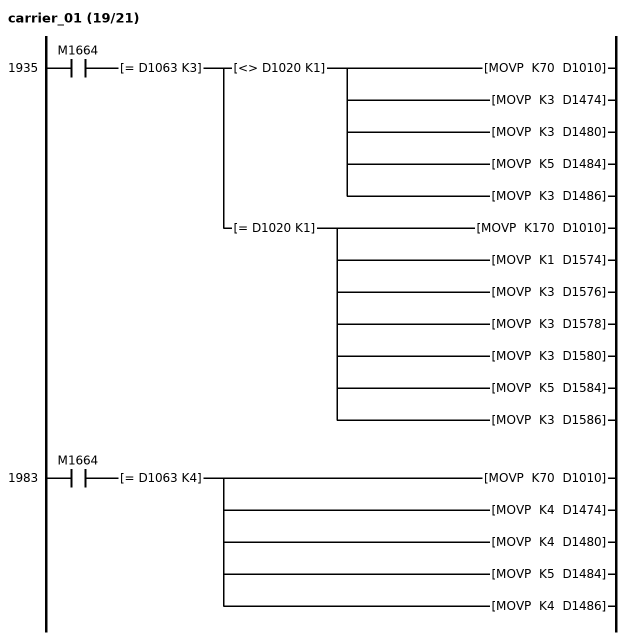
1935  LD      M1664
      AND=    D1063 K3
      MPS
      AND<>   D1020 K1
      MOVP    K70 D1010
      MOVP    K3 D1474
      MOVP    K3 D1480
      MOVP    K5 D1484
      MOVP    K3 D1486
      MPP
      AND=    D1020 K1
      MOVP    K170 D1010
      MOVP    K1 D1574
      MOVP    K3 D1576
      MOVP    K3 D1578
      MOVP    K3 D1580
      MOVP    K5 D1584
      MOVP    K3 D1586
1983  LD      M1664
      AND=    D1063 K4
      MOVP    K70 D1010
      MOVP    K4 D1474
      MOVP    K4 D1480
      MOVP    K5 D1484
      MOVP    K4 D1486
